{attribute 'GeneratedUsingTerminal: EL3356-0000-0017'}
{attribute addProperty BoxType "EL3356-0000-0017"}
{attribute addProperty Id "CtrlAT %Q*Ctrl_AEDC374E4"}
{attribute addProperty CRC "1234677494"}
{attribute addProperty Size "4"}
TYPE RMB_Control_4997AEF6 EXTENDS OutputBase_10CEE7DE :
STRUCT
	{attribute addProperty Name "Ctrl"}
	Ctrl AT %Q* : Ctrl_AEDC374E;
END_STRUCT
END_TYPE

(* stored: Version 1.2.0.0, ProductVersion 3.1.4024.11
   DUT RMB_Control_4997AEF6: Id {c17ef411-7836-43e4-b9ec-e1a067a37cfe} *)
